PROGRAM MAIN
VAR
END_VAR

END_PROGRAM

(* stored: Version 1.1.0.1, ProductVersion 3.1.4024.10
   POU MAIN: Id {36816d8f-5e91-4416-a7bc-947fc4f27113}, SpecialFunc None *)
